// TIA Portal V18 export
VAR_GLOBAL   // PLC tag table "TestResult"
END_VAR
VAR_GLOBAL CONSTANT   // user constants
   VacuumTestOK : Int := 1;
   VacuumTestNG : Int := 2;
   NitTestNG : Int := 2;
   NitTestOK : Int := 1;
END_VAR
